(* Logix 5000 project; controller MaquinaDeRechazo Emulate 5570 rev 32.11; software revision 32.00 *)

TASK MainTask (continuous, watchdog 500 ms) : MainProgram

MODULES
   Local : Emulate 5570 (ICP 2, rev 32.11)
END_MODULES

VAR_GLOBAL   (* controller tags *)
   BotOK : BOOL;
   BotOK_Off : BOOL;
   BotRe : BOOL;
   BotRe_Off : BOOL;
   Bottle_Counter : COUNTER := (PRE := 35, DN := 1);
   Bottle_Reject : COUNTER := (PRE := 20);
   Cilindro : BOOL;
   Conveyor1 : BOOL := 1;
   Conveyor2 : BOOL;
   E0 : BOOL;
   E1_Preparar : BOOL;
   E2_Transportar : BOOL := 1;
   E3_Decidir : BOOL;
   E4_Rechazar : BOOL;
   E5_PermitirPaso : BOOL;
   E6_Conteo : BOOL;
   E7_Finalizar : BOOL;
   ESTOP_OK : BOOL := 1;
   GUARDAS_OK : BOOL := 1;
   M1 : BOOL;
   ND_BotOK : DINT;
   ND_BotOK_H : BOOL;
   ND_BotOK_HH : BOOL;
   ND_BotOK_L : BOOL;
   ND_BotOK_LL : BOOL;
   ND_BotRe : DINT;
   ND_BotRe_H : BOOL;
   ND_BotRe_HH : BOOL;
   ND_BotRe_L : BOOL;
   ND_BotRe_LL : BOOL;
   ND_LoteMalo : BOOL;
   ND_ResConteo : BOOL;
   PB_START : BOOL;
   PB_STOP : BOOL;
   S_BOTELLA_INACEPTABLE : BOOL;
   S_BOTELLA_INSPECCION : BOOL;
   S_BOTELLA_OK : BOOL;
   S_HOME_RECHAZO : BOOL := 1;
   S_SALIDA_CONFIRMADA : BOOL;
   S_SALIDA_RECHAZO : BOOL;
   SIN_FALLAS : BOOL := 1;
   V1 : BOOL;
END_VAR

PROGRAM MainProgram   (* main routine MainRoutine *)

ROUTINE MainRoutine   (* ladder *)
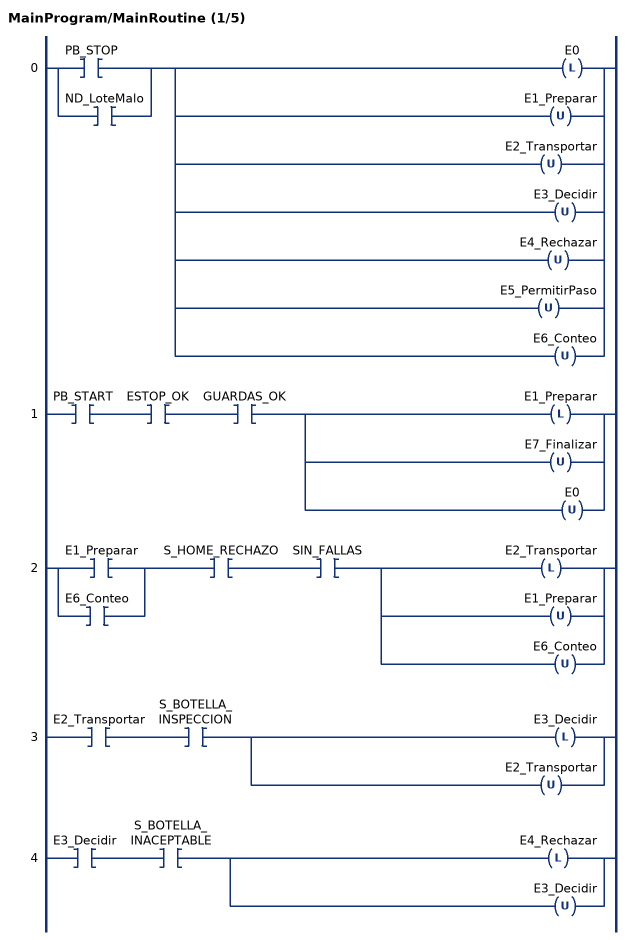
   0: [XIC(PB_STOP) ,XIC(ND_LoteMalo) ][OTL(E0) ,[OTU(E1_Preparar) ,[OTU(E2_Transportar) ,[OTU(E3_Decidir) ,[OTU(E4_Rechazar) ,[OTU(E5_PermitirPaso) ,OTU(E6_Conteo) ] ] ] ] ] ];
   1: XIC(PB_START)XIC(ESTOP_OK)XIC(GUARDAS_OK)[OTL(E1_Preparar) ,[OTU(E7_Finalizar) ,OTU(E0) ] ];
   2: [XIC(E1_Preparar) ,XIC(E6_Conteo) ]XIC(S_HOME_RECHAZO)XIC(SIN_FALLAS)[OTL(E2_Transportar) ,[OTU(E1_Preparar) ,OTU(E6_Conteo) ] ];
   3: XIC(E2_Transportar)XIC(S_BOTELLA_INSPECCION)[OTL(E3_Decidir) ,OTU(E2_Transportar) ];
   4: XIC(E3_Decidir)XIC(S_BOTELLA_INACEPTABLE)[OTL(E4_Rechazar) ,OTU(E3_Decidir) ];
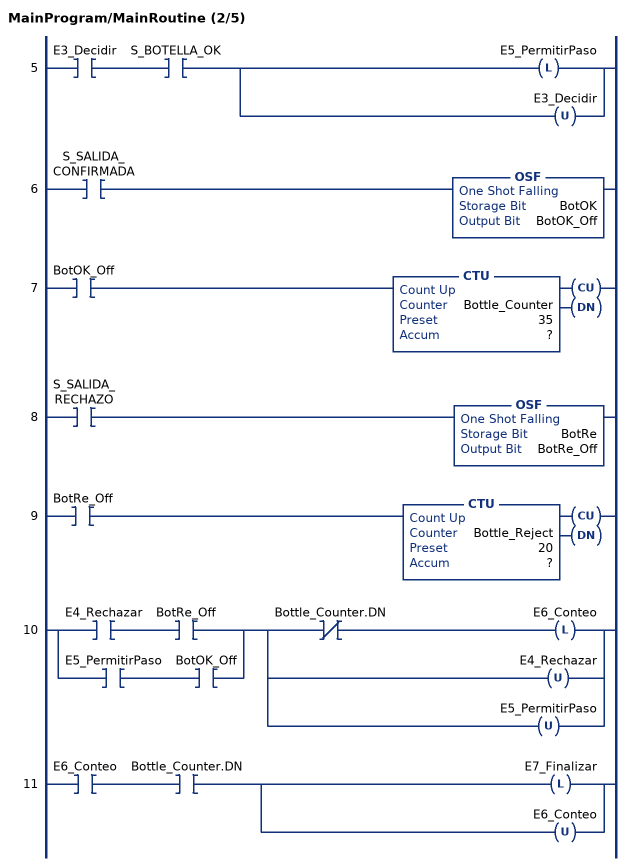
   5: XIC(E3_Decidir)XIC(S_BOTELLA_OK)[OTL(E5_PermitirPaso) ,OTU(E3_Decidir) ];
   6: XIC(S_SALIDA_CONFIRMADA)OSF(BotOK,BotOK_Off);
   7: XIC(BotOK_Off)CTU(Bottle_Counter,?,?);
   8: XIC(S_SALIDA_RECHAZO)OSF(BotRe,BotRe_Off);
   9: XIC(BotRe_Off)CTU(Bottle_Reject,?,?);
   10: [XIC(E4_Rechazar) XIC(BotRe_Off) ,XIC(E5_PermitirPaso) XIC(BotOK_Off) ][XIO(Bottle_Counter.DN) OTL(E6_Conteo) ,[OTU(E4_Rechazar) ,OTU(E5_PermitirPaso) ] ];
   11: XIC(E6_Conteo)XIC(Bottle_Counter.DN)[OTL(E7_Finalizar) ,OTU(E6_Conteo) ];
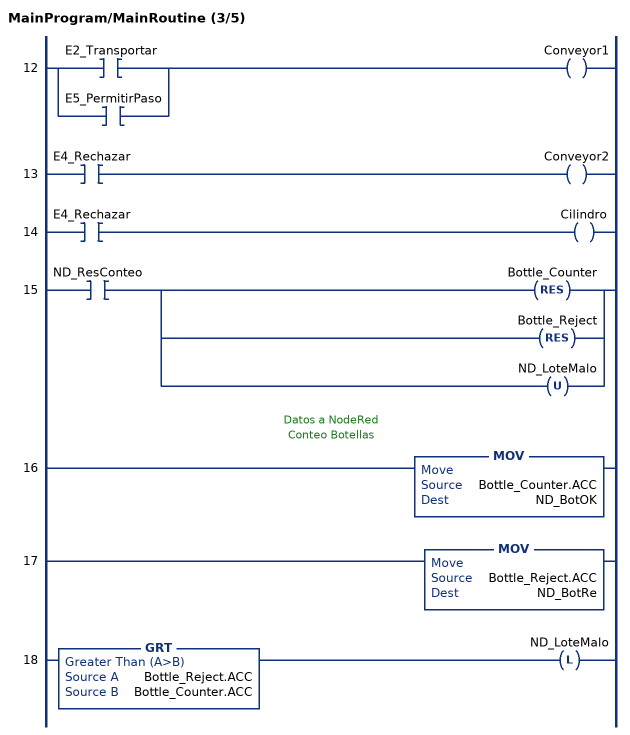
   12: [XIC(E2_Transportar) ,XIC(E5_PermitirPaso) ]OTE(Conveyor1);
   13: XIC(E4_Rechazar)OTE(Conveyor2);
   14: XIC(E4_Rechazar)OTE(Cilindro);
   15: XIC(ND_ResConteo)[RES(Bottle_Counter) ,[RES(Bottle_Reject) ,OTU(ND_LoteMalo) ] ];
   // Datos a NodeRed
   // Conteo Botellas
   16: MOV(Bottle_Counter.ACC,ND_BotOK);
   17: MOV(Bottle_Reject.ACC,ND_BotRe);
   18: GRT(Bottle_Reject.ACC,Bottle_Counter.ACC)OTL(ND_LoteMalo);
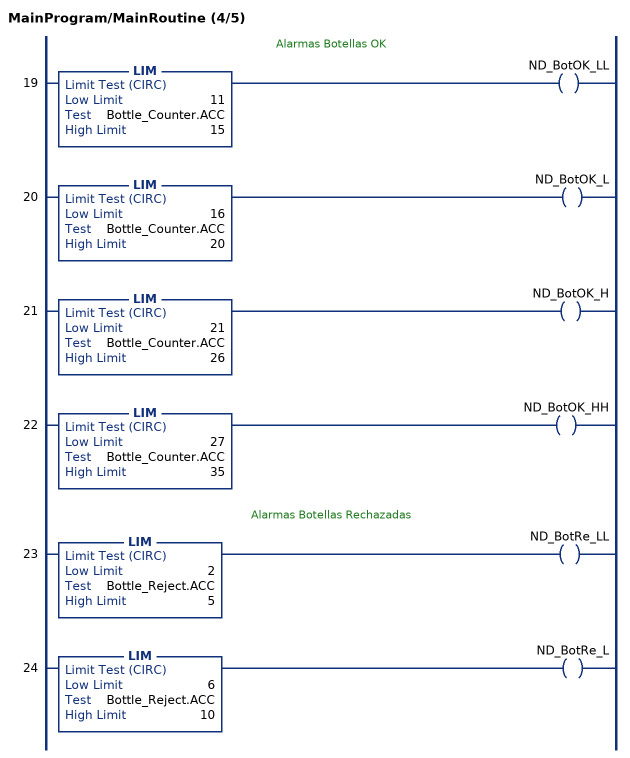
   // Alarmas Botellas OK
   19: LIM(11,Bottle_Counter.ACC,15)OTE(ND_BotOK_LL);
   20: LIM(16,Bottle_Counter.ACC,20)OTE(ND_BotOK_L);
   21: LIM(21,Bottle_Counter.ACC,26)OTE(ND_BotOK_H);
   22: LIM(27,Bottle_Counter.ACC,35)OTE(ND_BotOK_HH);
   // Alarmas Botellas Rechazadas
   23: LIM(2,Bottle_Reject.ACC,5)OTE(ND_BotRe_LL);
   24: LIM(6,Bottle_Reject.ACC,10)OTE(ND_BotRe_L);
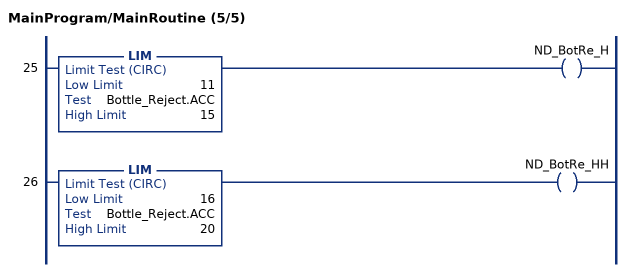
   25: LIM(11,Bottle_Reject.ACC,15)OTE(ND_BotRe_H);
   26: LIM(16,Bottle_Reject.ACC,20)OTE(ND_BotRe_HH);
END_ROUTINE
END_PROGRAM
